FUNCTION_BLOCK FB_ReceivePower_Left
VAR_IN_OUT
	Inputs_Left : CANRXQUEUESTRUCT_E_32;
	Outputs_Left : CANTXQUEUESTRUCT_E_32;
END_VAR
VAR_OUTPUT
	Power_Left : LREAL;
	JpM_Left : LREAL;
END_VAR
VAR
	MessageReceived : ARRAY[0..31] OF EXTCANQUEUE;
	i : INT;
	fbPPS_Timer : TON;
	nPacketsPerSecond: INT;
	nReceiveCounter : INT;
	nLastReceiveCounter : INT;
	
END_VAR

FOR i := 0 TO (Inputs_Left.NoOfRxMessages-1) DO
    IF Inputs_Left.RxMessages[i].cobId = 1700 THEN  
     	Power_Left := INT_TO_LREAL(DWORD_TO_INT(SHL(USINT_TO_UDINT(Inputs_Left.RxMessages[i].data[0]), 24) OR SHL(USINT_TO_UDINT(Inputs_Left.RxMessages[i].data[1]), 16) OR SHL(USINT_TO_UDINT(Inputs_Left.RxMessages[i].data[2]), 8)  OR USINT_TO_UDINT(Inputs_Left.RxMessages[i].data[3]))) / 100.0;
		JpM_Left := INT_TO_LREAL(DWORD_TO_INT(SHL(USINT_TO_UDINT(Inputs_Left.RxMessages[i].data[4]), 24) OR SHL(USINT_TO_UDINT(Inputs_Left.RxMessages[i].data[5]), 16) OR SHL(USINT_TO_UDINT(Inputs_Left.RxMessages[i].data[6]), 8)  OR USINT_TO_UDINT(Inputs_Left.RxMessages[i].data[7]))) / 100.0;
		
		nReceiveCounter := nReceiveCounter + 1;
    END_IF
END_FOR
fbPPS_Timer(IN := NOT fbPPS_Timer.Q, PT := T#1S);
IF fbPPS_Timer.Q THEN
			nPacketsPerSecond   := nReceiveCounter - nLastReceiveCounter;
			nLastReceiveCounter := nReceiveCounter;
END_IF

END_FUNCTION_BLOCK

(* stored: Version 1.1.0.1
   POU FB_ReceivePower_Left: Id {607bc68a-bc9e-41d0-b1ac-edad311bc77b}, SpecialFunc None *)
